// TIA Portal V18 export
DATA_BLOCK "AHUDI"   // DB113
{ S7_Optimized_Access := 'FALSE' }
VERSION : 0.1
// stored: AutoNumber false, DBAccessibleFromOPCUA true, IsOnlyStoredInLoadMemory false, IsWriteProtectedInAS false
   VAR RETAIN
      DI { S7_SetPoint := 'True'} : "UDT_AHUsDI";
   END_VAR
BEGIN
END_DATA_BLOCK
